// TIA Portal V20 export
// export: Created 2026-07-10T11:12:27.6439325Z, ExportSetting WithDefaults, DisplayName Totally Integrated Automation Portal, DisplayVersion V20, DisplayName TIA Portal Openness, DisplayVersion V20, DisplayName TIA Portal Version Control Interface, DisplayVersion V20, DisplayName STEP 7 Professional, DisplayVersion V20, DisplayName STEP 7 Safety, DisplayVersion V20, DisplayName WinCC Basic/Comfort/Advanced, DisplayVersion V20, DisplayName WinCC Unified, DisplayVersion V20
DATA_BLOCK "Dampers_DB"   // DB9
VERSION : 0.1
// stored: AutoNumber true, DBAccessibleFromOPCUA true, InstanceOfName Dampers, InstanceOfType FB
"Dampers"
   // VAR
   //    DamperController1 { S7_SetPoint := 'True'} : "DamperController";
   //    DamperController2 { S7_SetPoint := 'True'} : "DamperController";
   //    DamperController3 { S7_SetPoint := 'True'} : "DamperController";
   // END_VAR
BEGIN
   DamperController1.ManualMode := TRUE;
   DamperController1.ManaulOpen := FALSE;
   DamperController1.ManualClose := TRUE;
   DamperController1.TankLevel := 0.0;
   DamperController1.TankLevelSetpoint := 100.25;
   DamperController1.TankLevelMin := 200.5;
   DamperController1.TankLevelMax := 0.0;
   DamperController1.UsePID := FALSE;
   DamperController1.PID_DeadZone := 0.0;
   DamperController1.PID_KP := 0.0;
   DamperController1.PID_KI := 0.0;
   DamperController1.PID_KD := 0.0;
   DamperController1.PID_TI := 0.0;
   DamperController1.LimitSwitch0 := FALSE;
   DamperController1.LimitSwitch100 := FALSE;
   DamperController1.PouseMove := 5;
   DamperController1.PositionDeadzone := 0.0;
   DamperController1.StartAjustment := FALSE;
   DamperController1.CancelAjustment := FALSE;
   DamperController1.ResetPosition := FALSE;
   DamperController1.Open := FALSE;
   DamperController1.Close := FALSE;
   DamperController1.CurrentPosition := 0.0;
   DamperController1.PositionError := FALSE;
   DamperController1.PositionSetPoint := 100.0;
   DamperController1.AdjustBusy := FALSE;
   DamperController1.AdjustError := FALSE;
   DamperController1.FullMovingTime := 0.0;
   DamperController1.MoveToLimitSwitch := FALSE;
   DamperController1.AdjustmentDone := 16#0000;
   DamperController1.LappedSetpoint := 100.0;
   DamperController1.isMoving := FALSE;
   DamperController1.isAutoMode := FALSE;
   DamperController1.isReady := FALSE;
   DamperController1.EnablePIDTON.PT := T#0MS;
   DamperController1.EnablePIDTON.IN := FALSE;
   DamperController1.PIDRegulator.Enable := FALSE;
   DamperController1.PIDRegulator.Tanklevel := 0.0;
   DamperController1.PIDRegulator.TankLevelSetpoint := 100.25;
   DamperController1.PIDRegulator.KP := 0.0;
   DamperController1.PIDRegulator.KI := 0.0;
   DamperController1.PIDRegulator.KD := 0.0;
   DamperController1.PIDRegulator.TI := T#0MS;
   DamperController1.PIDRegulator.LimitMin := 0.0;
   DamperController1.PIDRegulator.LimitMax := 100.0;
   DamperController1.PIDRegulator.DeadZone := 0.0;
   DamperController1.PIDRegulator.DamperPosition := 0.0;
   DamperController1.PIDRegulator."e" := 100.25;
   DamperController1.PIDRegulator.PValue := 0.0;
   DamperController1.PIDRegulator.IValue := 0.0;
   DamperController1.PIDRegulator.DValue := 0.0;
   DamperController1.PIDRegulator.init := TRUE;
   DamperController1.PIDRegulator.TopLevelSetPoint := 100.25;
   DamperController1.PIDRegulator.BottomlevelSetPoint := 100.25;
   DamperController1.PIDRegulator.PrevValue := 0.0;
   DamperController1.PIDRegulator.TON1.PT := T#0MS;
   DamperController1.PIDRegulator.TON1.IN := FALSE;
   DamperController1.HystRegulator.Enable := FALSE;
   DamperController1.HystRegulator.TankLevel := 0.0;
   DamperController1.HystRegulator.TankLevelMin := 200.5;
   DamperController1.HystRegulator.TankLevelMax := 0.0;
   DamperController1.HystRegulator.Open := FALSE;
   DamperController1.HystRegulator.Close := FALSE;
   DamperController1.HystRegulator.PositionSetpoint := 0.0;
   DamperController1.RepositionRTrig.CLK := FALSE;
   DamperController1.RepositionRTrig.Q := FALSE;
   DamperController1.RepositionRTrig.Stat_Bit := FALSE;
   DamperController1.MotorPositionNoFeedback.Enable := TRUE;
   DamperController1.MotorPositionNoFeedback.LimitSwitch0 := FALSE;
   DamperController1.MotorPositionNoFeedback.LimitSwitch100 := FALSE;
   DamperController1.MotorPositionNoFeedback.Invalidate := FALSE;
   DamperController1.MotorPositionNoFeedback.FullMovingTime := 0.0;
   DamperController1.MotorPositionNoFeedback.LappingZone := 1.0;
   DamperController1.MotorPositionNoFeedback.Open := FALSE;
   DamperController1.MotorPositionNoFeedback.Close := FALSE;
   DamperController1.MotorPositionNoFeedback.CurrentPosition := 0.0;
   DamperController1.MotorPositionNoFeedback.Error := FALSE;
   DamperController1.MotorPositionNoFeedback.PreviousPosition := 0.0;
   DamperController1.MotorPositionNoFeedback.OnePercentImpulse := 0.0;
   DamperController1.MotorPositionNoFeedback.MovingTimer1.PT := T#0MS;
   DamperController1.MotorPositionNoFeedback.MovingTimer1.IN := FALSE;
   DamperController1.MotorPositionNoFeedback.MovingTimer2.PT := T#0MS;
   DamperController1.MotorPositionNoFeedback.MovingTimer2.IN := FALSE;
   DamperController1.MotorController.Enable := FALSE;
   DamperController1.MotorController.CurrentPosition := 0.0;
   DamperController1.MotorController.SetpointPosition := 100.0;
   DamperController1.MotorController.PositionDeadzone := 0.0;
   DamperController1.MotorController.MinimalPulse := T#100MS;
   DamperController1.MotorController.PauseMode := T#5S;
   DamperController1.MotorController.isMoving := FALSE;
   DamperController1.MotorController.MoveNow := FALSE;
   DamperController1.MotorController.MinReversPause := T#2S;
   DamperController1.MotorController.PositionError := FALSE;
   DamperController1.MotorController.Open := FALSE;
   DamperController1.MotorController.Close := FALSE;
   DamperController1.MotorController.Opening := FALSE;
   DamperController1.MotorController.Closing := FALSE;
   DamperController1.MotorController.MovingTOF.PT := T#0MS;
   DamperController1.MotorController.MovingTOF.IN := FALSE;
   DamperController1.MotorController.OpeningTOF.PT := T#0MS;
   DamperController1.MotorController.OpeningTOF.IN := FALSE;
   DamperController1.MotorController.ClosingTOF.PT := T#0MS;
   DamperController1.MotorController.ClosingTOF.IN := FALSE;
   DamperController1.MotorController.TON1.PT := T#0MS;
   DamperController1.MotorController.TON1.IN := FALSE;
   DamperController1.MotorController.TON2.PT := T#0MS;
   DamperController1.MotorController.TON2.IN := FALSE;
   DamperController1.RepositionTON.PT := T#10S;
   DamperController1.RepositionTON.IN := TRUE;
   DamperController1.MotorMoverToSwitch.Enable := TRUE;
   DamperController1.MotorMoverToSwitch.Go := FALSE;
   DamperController1.MotorMoverToSwitch.TargetSwitch100 := FALSE;
   DamperController1.MotorMoverToSwitch.MovePause := T#5S;
   DamperController1.MotorMoverToSwitch.isMoving := FALSE;
   DamperController1.MotorMoverToSwitch.LimitSwitch0 := FALSE;
   DamperController1.MotorMoverToSwitch.LimitSwitch100 := FALSE;
   DamperController1.MotorMoverToSwitch.Open := FALSE;
   DamperController1.MotorMoverToSwitch.Close := FALSE;
   DamperController1.MotorMoverToSwitch.GoTo0 := FALSE;
   DamperController1.MotorMoverToSwitch.GoTo100 := FALSE;
   DamperController1.MotorMoverToSwitch.MovingTOF.PT := T#0MS;
   DamperController1.MotorMoverToSwitch.MovingTOF.IN := FALSE;
   DamperController1.MotorAdjustmentNoFeedback.Enable := FALSE;
   DamperController1.MotorAdjustmentNoFeedback.Start := FALSE;
   DamperController1.MotorAdjustmentNoFeedback.Cancel := FALSE;
   DamperController1.MotorAdjustmentNoFeedback.AbortTime := T#2M;
   DamperController1.MotorAdjustmentNoFeedback.MovePause := T#5S;
   DamperController1.MotorAdjustmentNoFeedback.isMoving := FALSE;
   DamperController1.MotorAdjustmentNoFeedback.LimitSwitch0 := FALSE;
   DamperController1.MotorAdjustmentNoFeedback.LimitSwitch100 := FALSE;
   DamperController1.MotorAdjustmentNoFeedback.Busy := FALSE;
   DamperController1.MotorAdjustmentNoFeedback.Error := FALSE;
   DamperController1.MotorAdjustmentNoFeedback.Open := FALSE;
   DamperController1.MotorAdjustmentNoFeedback.Close := FALSE;
   DamperController1.MotorAdjustmentNoFeedback.Done := 16#0000;
   DamperController1.MotorAdjustmentNoFeedback.FullMovingTime := 0.0;
   DamperController1.MotorAdjustmentNoFeedback."step" := 16#0000;
   DamperController1.MotorAdjustmentNoFeedback.StartRTrig.CLK := FALSE;
   DamperController1.MotorAdjustmentNoFeedback.StartRTrig.Q := FALSE;
   DamperController1.MotorAdjustmentNoFeedback.StartRTrig.Stat_Bit := FALSE;
   DamperController1.MotorAdjustmentNoFeedback.CancelRTrig.CLK := FALSE;
   DamperController1.MotorAdjustmentNoFeedback.CancelRTrig.Q := FALSE;
   DamperController1.MotorAdjustmentNoFeedback.CancelRTrig.Stat_Bit := FALSE;
   DamperController1.MotorAdjustmentNoFeedback.MovingTOF.PT := T#0MS;
   DamperController1.MotorAdjustmentNoFeedback.MovingTOF.IN := FALSE;
   DamperController1.MotorAdjustmentNoFeedback.MovingTON.PT := T#0MS;
   DamperController1.MotorAdjustmentNoFeedback.MovingTON.IN := FALSE;
   DamperController1.MotorAdjustmentNoFeedback.PauseTON.PT := T#0MS;
   DamperController1.MotorAdjustmentNoFeedback.PauseTON.IN := FALSE;
   DamperController2.ManualMode := TRUE;
   DamperController2.ManaulOpen := FALSE;
   DamperController2.ManualClose := TRUE;
   DamperController2.TankLevel := 0.0;
   DamperController2.TankLevelSetpoint := 0.0;
   DamperController2.TankLevelMin := 0.0;
   DamperController2.TankLevelMax := 0.0;
   DamperController2.UsePID := FALSE;
   DamperController2.PID_DeadZone := 0.0;
   DamperController2.PID_KP := 0.0;
   DamperController2.PID_KI := 0.0;
   DamperController2.PID_KD := 0.0;
   DamperController2.PID_TI := 0.0;
   DamperController2.LimitSwitch0 := FALSE;
   DamperController2.LimitSwitch100 := FALSE;
   DamperController2.PouseMove := 5;
   DamperController2.PositionDeadzone := 0.0;
   DamperController2.StartAjustment := FALSE;
   DamperController2.CancelAjustment := FALSE;
   DamperController2.ResetPosition := FALSE;
   DamperController2.Open := FALSE;
   DamperController2.Close := FALSE;
   DamperController2.CurrentPosition := 0.0;
   DamperController2.PositionError := FALSE;
   DamperController2.PositionSetPoint := 0.0;
   DamperController2.AdjustBusy := FALSE;
   DamperController2.AdjustError := FALSE;
   DamperController2.FullMovingTime := 0.0;
   DamperController2.MoveToLimitSwitch := FALSE;
   DamperController2.AdjustmentDone := 16#0000;
   DamperController2.LappedSetpoint := 0.0;
   DamperController2.isMoving := FALSE;
   DamperController2.isAutoMode := FALSE;
   DamperController2.isReady := FALSE;
   DamperController2.EnablePIDTON.PT := T#0MS;
   DamperController2.EnablePIDTON.IN := FALSE;
   DamperController2.PIDRegulator.Enable := FALSE;
   DamperController2.PIDRegulator.Tanklevel := 0.0;
   DamperController2.PIDRegulator.TankLevelSetpoint := 0.0;
   DamperController2.PIDRegulator.KP := 0.0;
   DamperController2.PIDRegulator.KI := 0.0;
   DamperController2.PIDRegulator.KD := 0.0;
   DamperController2.PIDRegulator.TI := T#0MS;
   DamperController2.PIDRegulator.LimitMin := 0.0;
   DamperController2.PIDRegulator.LimitMax := 100.0;
   DamperController2.PIDRegulator.DeadZone := 0.0;
   DamperController2.PIDRegulator.DamperPosition := 0.0;
   DamperController2.PIDRegulator."e" := 0.0;
   DamperController2.PIDRegulator.PValue := 0.0;
   DamperController2.PIDRegulator.IValue := 0.0;
   DamperController2.PIDRegulator.DValue := 0.0;
   DamperController2.PIDRegulator.init := TRUE;
   DamperController2.PIDRegulator.TopLevelSetPoint := 0.0;
   DamperController2.PIDRegulator.BottomlevelSetPoint := 0.0;
   DamperController2.PIDRegulator.PrevValue := 0.0;
   DamperController2.PIDRegulator.TON1.PT := T#0MS;
   DamperController2.PIDRegulator.TON1.IN := FALSE;
   DamperController2.HystRegulator.Enable := FALSE;
   DamperController2.HystRegulator.TankLevel := 0.0;
   DamperController2.HystRegulator.TankLevelMin := 0.0;
   DamperController2.HystRegulator.TankLevelMax := 0.0;
   DamperController2.HystRegulator.Open := FALSE;
   DamperController2.HystRegulator.Close := FALSE;
   DamperController2.HystRegulator.PositionSetpoint := 0.0;
   DamperController2.RepositionRTrig.CLK := FALSE;
   DamperController2.RepositionRTrig.Q := FALSE;
   DamperController2.RepositionRTrig.Stat_Bit := FALSE;
   DamperController2.MotorPositionNoFeedback.Enable := TRUE;
   DamperController2.MotorPositionNoFeedback.LimitSwitch0 := FALSE;
   DamperController2.MotorPositionNoFeedback.LimitSwitch100 := FALSE;
   DamperController2.MotorPositionNoFeedback.Invalidate := FALSE;
   DamperController2.MotorPositionNoFeedback.FullMovingTime := 0.0;
   DamperController2.MotorPositionNoFeedback.LappingZone := 1.0;
   DamperController2.MotorPositionNoFeedback.Open := FALSE;
   DamperController2.MotorPositionNoFeedback.Close := FALSE;
   DamperController2.MotorPositionNoFeedback.CurrentPosition := 0.0;
   DamperController2.MotorPositionNoFeedback.Error := FALSE;
   DamperController2.MotorPositionNoFeedback.PreviousPosition := 0.0;
   DamperController2.MotorPositionNoFeedback.OnePercentImpulse := 0.0;
   DamperController2.MotorPositionNoFeedback.MovingTimer1.PT := T#0MS;
   DamperController2.MotorPositionNoFeedback.MovingTimer1.IN := FALSE;
   DamperController2.MotorPositionNoFeedback.MovingTimer2.PT := T#0MS;
   DamperController2.MotorPositionNoFeedback.MovingTimer2.IN := FALSE;
   DamperController2.MotorController.Enable := FALSE;
   DamperController2.MotorController.CurrentPosition := 0.0;
   DamperController2.MotorController.SetpointPosition := 0.0;
   DamperController2.MotorController.PositionDeadzone := 0.0;
   DamperController2.MotorController.MinimalPulse := T#100MS;
   DamperController2.MotorController.PauseMode := T#5S;
   DamperController2.MotorController.isMoving := FALSE;
   DamperController2.MotorController.MoveNow := FALSE;
   DamperController2.MotorController.MinReversPause := T#2S;
   DamperController2.MotorController.PositionError := FALSE;
   DamperController2.MotorController.Open := FALSE;
   DamperController2.MotorController.Close := FALSE;
   DamperController2.MotorController.Opening := FALSE;
   DamperController2.MotorController.Closing := FALSE;
   DamperController2.MotorController.MovingTOF.PT := T#0MS;
   DamperController2.MotorController.MovingTOF.IN := FALSE;
   DamperController2.MotorController.OpeningTOF.PT := T#0MS;
   DamperController2.MotorController.OpeningTOF.IN := FALSE;
   DamperController2.MotorController.ClosingTOF.PT := T#0MS;
   DamperController2.MotorController.ClosingTOF.IN := FALSE;
   DamperController2.MotorController.TON1.PT := T#0MS;
   DamperController2.MotorController.TON1.IN := FALSE;
   DamperController2.MotorController.TON2.PT := T#0MS;
   DamperController2.MotorController.TON2.IN := FALSE;
   DamperController2.RepositionTON.PT := T#10S;
   DamperController2.RepositionTON.IN := TRUE;
   DamperController2.MotorMoverToSwitch.Enable := TRUE;
   DamperController2.MotorMoverToSwitch.Go := FALSE;
   DamperController2.MotorMoverToSwitch.TargetSwitch100 := FALSE;
   DamperController2.MotorMoverToSwitch.MovePause := T#5S;
   DamperController2.MotorMoverToSwitch.isMoving := FALSE;
   DamperController2.MotorMoverToSwitch.LimitSwitch0 := FALSE;
   DamperController2.MotorMoverToSwitch.LimitSwitch100 := FALSE;
   DamperController2.MotorMoverToSwitch.Open := FALSE;
   DamperController2.MotorMoverToSwitch.Close := FALSE;
   DamperController2.MotorMoverToSwitch.GoTo0 := FALSE;
   DamperController2.MotorMoverToSwitch.GoTo100 := FALSE;
   DamperController2.MotorMoverToSwitch.MovingTOF.PT := T#0MS;
   DamperController2.MotorMoverToSwitch.MovingTOF.IN := FALSE;
   DamperController2.MotorAdjustmentNoFeedback.Enable := FALSE;
   DamperController2.MotorAdjustmentNoFeedback.Start := FALSE;
   DamperController2.MotorAdjustmentNoFeedback.Cancel := FALSE;
   DamperController2.MotorAdjustmentNoFeedback.AbortTime := T#2M;
   DamperController2.MotorAdjustmentNoFeedback.MovePause := T#5S;
   DamperController2.MotorAdjustmentNoFeedback.isMoving := FALSE;
   DamperController2.MotorAdjustmentNoFeedback.LimitSwitch0 := FALSE;
   DamperController2.MotorAdjustmentNoFeedback.LimitSwitch100 := FALSE;
   DamperController2.MotorAdjustmentNoFeedback.Busy := FALSE;
   DamperController2.MotorAdjustmentNoFeedback.Error := FALSE;
   DamperController2.MotorAdjustmentNoFeedback.Open := FALSE;
   DamperController2.MotorAdjustmentNoFeedback.Close := FALSE;
   DamperController2.MotorAdjustmentNoFeedback.Done := 16#0000;
   DamperController2.MotorAdjustmentNoFeedback.FullMovingTime := 0.0;
   DamperController2.MotorAdjustmentNoFeedback."step" := 16#0000;
   DamperController2.MotorAdjustmentNoFeedback.StartRTrig.CLK := FALSE;
   DamperController2.MotorAdjustmentNoFeedback.StartRTrig.Q := FALSE;
   DamperController2.MotorAdjustmentNoFeedback.StartRTrig.Stat_Bit := FALSE;
   DamperController2.MotorAdjustmentNoFeedback.CancelRTrig.CLK := FALSE;
   DamperController2.MotorAdjustmentNoFeedback.CancelRTrig.Q := FALSE;
   DamperController2.MotorAdjustmentNoFeedback.CancelRTrig.Stat_Bit := FALSE;
   DamperController2.MotorAdjustmentNoFeedback.MovingTOF.PT := T#0MS;
   DamperController2.MotorAdjustmentNoFeedback.MovingTOF.IN := FALSE;
   DamperController2.MotorAdjustmentNoFeedback.MovingTON.PT := T#0MS;
   DamperController2.MotorAdjustmentNoFeedback.MovingTON.IN := FALSE;
   DamperController2.MotorAdjustmentNoFeedback.PauseTON.PT := T#0MS;
   DamperController2.MotorAdjustmentNoFeedback.PauseTON.IN := FALSE;
END_DATA_BLOCK
